// TwinCAT 3 PLC project Dyanmisch_Converteren
// ProgramVersion: 3.1.4024.0
// libraries:
//   Tc2_Standard, * (Beckhoff Automation GmbH)
//   Tc2_System, * (Beckhoff Automation GmbH)
//   Tc3_Module, * (Beckhoff Automation GmbH)
// project tree:
//   / PlcTask.TcTTO
//   POUs/ MAIN.TcPOU
// (motion and I/O tree: see PLC project potentiometer_inlezen)
// real-time tasks:
//   TASK PlcTask: cycle T#10ms, priority 20, ADS port 350
//   TASK PlcTask1: cycle T#10ms, priority 21, ADS port 351
//   TASK PlcTask2: cycle T#10ms, priority 22, ADS port 352
//   TASK PlcTask3: cycle T#10ms, priority 26, ADS port 353
//   TASK PlcTask4: cycle T#10ms, priority 25, ADS port 354
//   TASK PlcTask5: cycle T#10ms, priority 24, ADS port 355
//   TASK PlcTask6: cycle T#10ms, priority 23, ADS port 356
//   TASK PlcTask7: cycle T#10ms, priority 27, ADS port 357

CONFIGURATION Dyanmisch_Converteren
    RESOURCE PLC ON TwinCAT3
        TASK PlcTask(INTERVAL := T#10ms, PRIORITY := 21);
        PROGRAM MAIN WITH PlcTask : MAIN;
    END_RESOURCE
END_CONFIGURATION

// ---- POUs/MAIN.TcPOU
PROGRAM MAIN
VAR
	Waarde: BYTE;
	nScaledMax: INT := 10;
	potentiometer: INT;
END_VAR

(*
Declareer een variabele van het type INT, met de naam nScaledMax en een initial value van 10. Gebruik hiervoor de Auto Declare functie (zie afbeelding). 
Vervolgens schrijf je de code om de potentiometer-waarde te verschalen naar een getal tussen 0 en nScaledMax.
*)

Waarde:=LREAL_TO_BYTE(nScaledMax*(potentiometer/32767.0));

END_PROGRAM
